PROGRAM DebugMode
VAR
(* Common*)
	d_state: DINT;(*PowerOffState*)
	InitDone:BOOL;
	Busy: BOOL;
	fb_ton: TON;
	PowerState: INT;(*PowerOnState*)
	ton_t: TON;
(*Key Command*)
	LeftTopLinPositionNew:LREAL;
	LeftTopLinVelocityNew:LREAL:=0.02;
	btn_LeftTopLinMove:BOOL;
	btn_LeftTopLinStop:BOOL;
	RightTopLinPositionNew:LREAL;
	RightTopLinVelocityNew:LREAL:=0.02;
	btn_RightTopLinMove:BOOL;
	btn_RightTopLinStop:BOOL;
	LeftBottomLinPositionNew:LREAL;
	LeftBottomLinVelocityNew:LREAL:=0.02;
	btn_LeftBottomLinMove:BOOL;
	btn_LeftBottomLinStop:BOOL;
	RightBottomLinPositionNew:LREAL;
	RightBottomLinVelocityNew:LREAL:=0.02;
	btn_RightBottomLinMove:BOOL;
	btn_RightBottomLinStop:BOOL;
(*LeftTopLin*)
	fb_ton1_1:TON;
	fb_ton1_2:TON;
	LeftTopLinState:DINT;
	LeftTopLinBusy:BOOL;
	LeftTopLin_m_state: DINT;
	LeftTopLin_s_state: DINT;
(*RightTopLin*)
	fb_ton2_1:TON;
	fb_ton2_2:TON;
	RightTopLinState:DINT;
	RightTopLinBusy:BOOL;
	RightTopLin_m_state: DINT;
	RightTopLin_s_state: DINT;
(*LeftBottomLin*)
	fb_ton3_1:TON;
	fb_ton3_2:TON;
	LeftBottomLinState:DINT;
	LeftBottomLinBusy:BOOL;
	LeftBottomLin_m_state: DINT;
	LeftBottomLin_s_state: DINT;
(*RightBottomLin*)
	fb_ton4_1:TON;
	fb_ton4_2:TON;
	RightBottomLinState:DINT;
	RightBottomLinBusy:BOOL;
	RightBottomLin_m_state: DINT;
	RightBottomLin_s_state: DINT;


	btn_LeftTopStop: BOOL;
	(*¼ì²âµ½ÏÞÎ»£¬»Ö¸´Move×´Ì¬*)
	FTrig_ReachLS: F_TRIG;
	FTrig_btn_GapMove: F_TRIG;
	
	RTrig_LeftTopMove:R_TRIG;
	RTrig_RightTopMove:R_TRIG;
	RTrig_LeftBottomMove:R_TRIG;
	RTrig_RightBottomMove:R_TRIG;
	
END_VAR

(*********************************************************************Monitor All Carrirt Position***********************************************)
A_MonitoringAllAxis();
(*********************************************************************A_PosDiffDetection***********************************************)
A_PosDiffDetection();
//
IF st_Power=1 THEN
	InitDone:=TRUE;
END_IF
(*********************************************************************btn_PowerOn************************************************************)
IF btn_Power AND st_Power=0 THEN
	btn_PowerOn:=TRUE;
	btn_Power:=FALSE;
END_IF
IF btn_Power AND st_Power=1 THEN
	btn_PowerOff:=TRUE;
	btn_Power:=FALSE;
END_IF
(*********************************************************************btn_PowerOn************************************************************)
IF btn_PowerOn THEN
	A_PowerOn();
END_IF
(****************************************************ESTOP***********************************************)
IF NOT btn_PowerOff THEN
	IF st_Power=1 AND st_Couple<>0THEN
		Error:=TRUE;
		ErrorID:=101;
		FB_PlcEmergencyStop();
		LED_Error:=TRUE;
	END_IF
END_IF

(*********************************************************************btn_PowerOff************************************************************)
IF btn_PowerOff THEN
	A_PowerOff();
END_IF

A_Motion();
A_CheckTargetPos();


(****************************MoveIndicator***************************)
IF Velo_LeftTopLin>0 THEN
	LeftTopLinMoveIndicator:=1;
ELSIF Velo_LeftTopLin<0 THEN
	LeftTopLinMoveIndicator:=-1;
ELSE
	LeftTopLinMoveIndicator:=0;
END_IF
IF Velo_RightTopLin>0 THEN
	RightTopLinMoveIndicator:=1;
ELSIF Velo_RightTopLin<0 THEN
	RightTopLinMoveIndicator:=-1;
ELSE
	RightTopLinMoveIndicator:=0;
END_IF
IF Velo_LeftBottomLin>0 THEN
	LeftBottomLinMoveIndicator:=1;
ELSIF Velo_LeftBottomLin<0 THEN
	LeftBottomLinMoveIndicator:=-1;
ELSE
	LeftBottomLinMoveIndicator:=0;
END_IF
IF Velo_RightBottomLin>0 THEN
	RightBottomLinMoveIndicator:=1;
ELSIF Velo_RightBottomLin<0 THEN
	RightBottomLinMoveIndicator:=-1;
ELSE
	RightBottomLinMoveIndicator:=0;
END_IF
(*********************************************************************ÏÞÎ»Åö´¥×´Ì¬»Ö¸´************************************************************)
(*Èç¹û¼ì²âµ½ÏØÏÞÎ»¿ª¹ØÏÂ½µÑØ£¬»Ö¸´Move×´Ì¬*)
FTrig_ReachLS(CLK:=Unreach_LS_Far AND Unreach_LS_Near);
IF FTrig_ReachLS.Q THEN
	btn_LeftTopLinStop:=TRUE;
	btn_RightTopLinStop:=TRUE;
	btn_LeftBottomLinStop:=TRUE;
	btn_RightBottomLinStop:=TRUE;
END_IF
IF btn_LeftTopLinStop THEN
	btn_RightTopLinStop:=TRUE;
END_IF
IF btn_RightTopLinStop THEN
	btn_LeftBottomLinStop:=TRUE;
END_IF
IF btn_LeftBottomLinStop THEN
	btn_RightBottomLinStop:=TRUE;
END_IF

IF NOT Unreach_LS_Far AND LeftTopLinPositionNew-Pos_LeftTopLin>0.0005 AND btn_LeftTopLinMove THEN
	btn_LeftTopLinStop:=TRUE;
END_IF
IF NOT Unreach_LS_Near AND RightTopLinPositionNew-Pos_RightTopLin<0.0005 AND btn_RightTopLinMove THEN
	btn_RightTopLinStop:=TRUE;
END_IF
IF NOT Unreach_LS_Far AND LeftBottomLinPositionNew-Pos_LeftBottomLin>0.0005 AND btn_LeftBottomLinMove THEN
	btn_LeftBottomLinStop:=TRUE;
END_IF
IF NOT Unreach_LS_Near AND RightBottomLinPositionNew-Pos_RightBottomLin<0.0005 AND btn_RightBottomLinMove THEN
	btn_RightBottomLinStop:=TRUE;
END_IF

ACTION A_CheckTargetPos:
RTrig_LeftTopMove(CLK:=btn_LeftTopLinMove);
IF RTrig_LeftTopMove.Q THEN
	IF NOT st_Power THEN
			ErrorID:=1501;
			Error:=TRUE;
			ErrorDescription:='Plz PowerOn Frist';
			LED_Error:=TRUE;
			//RETURN;
		ELSIF ABS(LeftTopLinPositionNew-Pos_LeftTopLin)>Threshold_LeftTopPos_Debug THEN
			btn_LeftTopLinStop:=TRUE;
			btn_LeftTopLinMove:=FALSE;
			ErrorID:=1502;
			Error:=TRUE;
			ErrorDescription:='targetPos Out of range!';
			LED_Error:=TRUE;
			//RETURN;
		ELSE
			ErrorID:=0;
			Error:=FALSE;
			ErrorDescription:='';
			LED_Error:=FALSE;
		END_IF
END_IF
RTrig_RightTopMove(CLK:=btn_RightTopLinMove);
IF RTrig_RightTopMove.Q THEN
	IF NOT st_Power THEN
			ErrorID:=1503;
			Error:=TRUE;
			ErrorDescription:='Plz PowerOn Frist';
			LED_Error:=TRUE;
			//RETURN;
		ELSIF ABS(RightTopLinPositionNew-Pos_RightTopLin)>Threshold_RightTopPos_Debug THEN
			btn_RightTopLinStop:=TRUE;
			btn_RightTopLinMove:=FALSE;
			ErrorID:=1504;
			Error:=TRUE;
			ErrorDescription:='targetPos Out of range!';
			LED_Error:=TRUE;
			//RETURN;
		ELSE
			ErrorID:=0;
			Error:=FALSE;
			ErrorDescription:='';
			LED_Error:=FALSE;
		END_IF
END_IF
RTrig_LeftBottomMove(CLK:=btn_LeftBottomLinMove);
IF RTrig_LeftBottomMove.Q THEN
	IF NOT st_Power THEN
			ErrorID:=1505;
			Error:=TRUE;
			ErrorDescription:='Plz PowerOn Frist';
			LED_Error:=TRUE;
			//RETURN;
		ELSIF ABS(LeftBottomLinPositionNew-Pos_LeftBottomLin)>Threshold_LeftBottomPos_Debug THEN
			btn_LeftBottomLinStop:=TRUE;
			btn_LeftBottomLinMove:=FALSE;
			ErrorID:=1506;
			Error:=TRUE;
			ErrorDescription:='targetPos Out of range!';
			LED_Error:=TRUE;
			//RETURN;
		ELSE
			ErrorID:=0;
			Error:=FALSE;
			ErrorDescription:='';
			LED_Error:=FALSE;
		END_IF
END_IF
RTrig_RightBottomMove(CLK:=btn_RightBottomLinMove);
IF RTrig_RightBottomMove.Q THEN
	IF NOT st_Power THEN
			ErrorID:=1507;
			Error:=TRUE;
			ErrorDescription:='Plz PowerOn Frist';
			LED_Error:=TRUE;
			//RETURN;
		ELSIF ABS(RightBottomLinPositionNew-Pos_RightBottomLin)>Threshold_RightBottomPos_Debug THEN
			btn_RightBottomLinStop:=TRUE;
			btn_RightBottomLinMove:=FALSE;
			ErrorID:=1508;
			Error:=TRUE;
			ErrorDescription:='targetPos Out of range!';
			LED_Error:=TRUE;
			//RETURN;
		ELSE
			ErrorID:=0;
			Error:=FALSE;
			ErrorDescription:='';
			LED_Error:=FALSE;
		END_IF
END_IF
END_ACTION

ACTION A_monitoringAllAxis:
(****************************************************************
NAME:			A_MonitoringAllAxis
DATA:			2017.5.8
VERSION:		1.0.0
DESCRIPTION:	

HISTORY:
				2017.5.8	NEW

***************************************************************)

(******************************************************************************************************************************************************)
IF st_power<>0 THEN

IF ABS(Pos_LeftTopLin-Pos_LeftBottomLin)>Threshold_LeftPos_Debug  THEN
		btn_LeftTopLinStop:=TRUE;
		btn_RightTopLinStop:=TRUE;
		btn_LeftBottomLinStop:=TRUE;
		btn_RightBottomLInStop:=TRUE;
		FB_PlcEmergencyStop();
		Error:=TRUE;
		ErrorID:=11;
		LED_Error:=TRUE;
END_IF

IF ABS(Pos_RightTopLin-Pos_RightBottomLin)>Threshold_RightPos_Debug  THEN
		btn_LeftTopLinStop:=TRUE;
		btn_RightTopLinStop:=TRUE;
		btn_LeftBottomLinStop:=TRUE;
		btn_RightBottomLInStop:=TRUE;
		FB_PlcEmergencyStop();
		Error:=TRUE;
		ErrorID:=12;
		LED_Error:=TRUE;
END_IF

IF ABS(Pos_LeftTopLin-Pos_RightTopLin)>Threshold_TopPos_Debug  THEN
		btn_LeftTopLinStop:=TRUE;
		btn_RightTopLinStop:=TRUE;
		btn_LeftBottomLinStop:=TRUE;
		btn_RightBottomLInStop:=TRUE;
		FB_PlcEmergencyStop();
		Error:=TRUE;
		ErrorID:=13;
		LED_Error:=TRUE;
END_IF

IF ABS(Pos_LeftBottomLin-Pos_RightBottomLin)>Threshold_BottomPos_Debug  THEN
		btn_LeftTopLinStop:=TRUE;
		btn_RightTopLinStop:=TRUE;
		btn_LeftBottomLinStop:=TRUE;
		btn_RightBottomLInStop:=TRUE;
		FB_PlcEmergencyStop();
		Error:=TRUE;
		ErrorID:=14;
		LED_Error:=TRUE;
END_IF
END_IF
(*********************************************************************************3.Ã¿Öá¹âÕ¤ºÍ±àÂëÆ÷Î»ÖÃ¶Ô±È¼ì²é**********************************************************************)
END_ACTION

ACTION A_Motion:
(*********************************************************************LeftTop_MOVE*****************************************************************)
//IF InitDone THEN
	IF btn_LeftTopLinMove THEN
		CASE LeftTopLin_m_state OF
			0:
				FB_Move.Mode:=4;					
				FB_Move.CoupleState:=st_Couple;
				FB_Move.PowerState:=st_Power;		
				FB_Move.LeftTopMove:=TRUE;			
				FB_Move.LeftTopPosition:=LeftTopLinPositionNew;
				FB_Move.LeftTopVelocity:=LeftTopLinVelocityNew;	
				FB_Move();								
				LeftTopLin_m_state:=1;
			1:
				FB_Move();
				IF NOT FB_Move.LeftTopDone THEN		
					LeftTopLin_m_state:=1;
					LED_Run:=TRUE;
				ELSE							
					LeftTopLin_m_state:=88;
				END_IF

			88:
				btn_LeftTopLinMove:=FALSE;				
				LeftTopLin_m_state:=0;
				LED_Run:=FALSE;
		END_CASE
	END_IF
//END_IF
(*******************************************************************LeftTop_STOP********************************************************************)
IF btn_LeftTopLinStop OR btn_reset THEN
	LED_Run:=FALSE;
	FB_Move.LeftTopReset:=TRUE;							
	FB_Move();										
	btn_LeftTopLinMove:=FALSE;						
	LeftTopLin_m_state:=0;										
	CASE LeftTopLin_s_state OF
			0:
				FB_Stop.Mode:=4;							
				FB_Stop.CoupleState:=st_Couple;			
				FB_Stop.PowerState:=st_Power;				
				FB_Stop.LeftTopStop:=TRUE;				
				FB_Stop();							
				LeftTopLin_s_state:=1;
			1:
				FB_Stop();
				IF NOT FB_Stop.LeftTopDone THEN		
					LeftTopLin_s_state:=1;
				ELSE								
					LeftTopLin_s_state:=88;
				END_IF
			88:
				btn_LeftTopLinStop:=FALSE;					
				FB_Move.LeftTopReset:=FALSE;				
				LeftTopLin_s_state:=0;
				btn_reset:=FALSE;
		END_CASE

END_IF
(*********************************************************************RightTop_MOVE*****************************************************************)
//IF InitDone THEN
	IF btn_RightTopLinMove THEN
		CASE RightTopLin_m_state OF
			0:
				FB_Move.Mode:=4;						
				FB_Move.CoupleState:=st_Couple;			
				FB_Move.PowerState:=st_Power;			
				FB_Move.RightTopMove:=TRUE;			
				FB_Move.RightTopPosition:=RightTopLinPositionNew;	
				FB_Move.RightTopVelocity:=RightTopLinVelocityNew;	
				FB_Move();								
				RightTopLin_m_state:=1;
			1:
				FB_Move();
				IF NOT FB_Move.RightTopDone THEN		
					RightTopLin_m_state:=1;
					LED_Run:=TRUE;
				ELSE								
					RightTopLin_m_state:=88;
				END_IF

			88:
				btn_RightTopLinMove:=FALSE;				
				RightTopLin_m_state:=0;
				LED_Run:=FALSE;
		END_CASE
	END_IF
//END_IF
(*******************************************************************RightTop_STOP********************************************************************)
IF btn_RightTopLinStop OR btn_reset THEN
	LED_Run:=FALSE;
	FB_Move.RightTopReset:=TRUE;						
	FB_Move();										
	btn_RightTopLinMove:=FALSE;							
	RightTopLin_m_state:=0;										
	CASE RightTopLin_s_state OF
			0:
				FB_Stop.Mode:=4;							
				FB_Stop.CoupleState:=st_Couple;		
				FB_Stop.PowerState:=st_Power;			
				FB_Stop.RightTopStop:=TRUE;				
				FB_Stop();							
				RightTopLin_s_state:=1;
			1:
				FB_Stop();
				IF NOT FB_Stop.RightTopDone THEN			
					RightTopLin_s_state:=1;
				ELSE								
					RightTopLin_s_state:=88;
				END_IF
			88:
				btn_RightTopLinStop:=FALSE;					
				FB_Move.RightTopReset:=FALSE;				
				RightTopLin_s_state:=0;
				btn_reset:=FALSE;
		END_CASE

END_IF
(*********************************************************************LeftBottom_MOVE*****************************************************************)
//IF InitDone THEN
	IF btn_LeftBottomLinMove THEN
		CASE LeftBottomLin_m_state OF
			0:
				FB_Move.Mode:=4;					
				FB_Move.CoupleState:=st_Couple;			
				FB_Move.PowerState:=st_Power;		
				FB_Move.LeftBottomMove:=TRUE;				(*Execute TRUE*)
				FB_Move.LeftBottomPosition:=LeftBottomLinPositionNew;	
				FB_Move.LeftBottomVelocity:=LeftBottomLinVelocityNew;
				FB_Move();								
				LeftBottomLin_m_state:=1;
			1:
				FB_Move();
				IF NOT FB_Move.LeftBottomDone THEN		
					LeftBottomLin_m_state:=1;
					LED_Run:=TRUE;
				ELSE								
					LeftBottomLin_m_state:=88;
				END_IF

			88:
				btn_LeftBottomLinMove:=FALSE;				
				LeftBottomLin_m_state:=0;
				LED_Run:=FALSE;
		END_CASE
	END_IF
//END_IF
(*******************************************************************LeftBottom_STOP********************************************************************)
IF btn_LeftBottomLinStop OR btn_reset THEN
	LED_Run:=FALSE;
	FB_Move.LeftBottomReset:=TRUE;						
	FB_Move();										
	btn_LeftBottomLinMove:=FALSE;						
	LeftBottomLin_m_state:=0;									
	CASE LeftBottomLin_s_state OF
			0:
				FB_Stop.Mode:=4;						
				FB_Stop.CoupleState:=st_Couple;		
				FB_Stop.PowerState:=st_Power;			
				FB_Stop.LeftBottomStop:=TRUE;				
				FB_Stop();						
				LeftBottomLin_s_state:=1;
			1:
				FB_Stop();
				IF NOT FB_Stop.LeftBottomDone THEN			
					LeftBottomLin_s_state:=1;
				ELSE								
					LeftBottomLin_s_state:=88;
				END_IF
			88:
				btn_LeftBottomLinStop:=FALSE;					
				FB_Move.LeftBottomReset:=FALSE;			
				LeftBottomLin_s_state:=0;
				btn_reset:=FALSE;
		END_CASE

END_IF

(*********************************************************************RightTop_MOVE*****************************************************************)
//IF InitDone THEN
	IF btn_RightBottomLinMove THEN
		CASE RightBottomLin_m_state OF
			0:
				FB_Move.Mode:=4;						
				FB_Move.CoupleState:=st_Couple;			
				FB_Move.PowerState:=st_Power;			
				FB_Move.RightBottomMove:=TRUE;				
				FB_Move.RightBottomPosition:=RightBottomLinPositionNew;	
				FB_Move.RightBottomVelocity:=RightBottomLinVelocityNew;	
				FB_Move();								
				RightBottomLin_m_state:=1;
			1:
				FB_Move();
				IF NOT FB_Move.RightBottomDone THEN			
					RightBottomLin_m_state:=1;
					LED_Run:=TRUE;
				ELSE									
					RightBottomLin_m_state:=88;
				END_IF

			88:
				btn_RightBottomLinMove:=FALSE;					
				RightBottomLin_m_state:=0;
				LED_Run:=FALSE;
		END_CASE
	END_IF
//END_IF
(*******************************************************************RightBottom_STOP********************************************************************)
IF btn_RightBottomLinStop OR btn_reset THEN
	LED_Run:=FALSE;
	FB_Move.RightBottomReset:=TRUE;							
	FB_Move();											
	btn_RightBottomLinMove:=FALSE;							
	RightBottomLin_m_state:=0;											
	CASE RightBottomLin_s_state OF
			0:
				FB_Stop.Mode:=4;							
				FB_Stop.CoupleState:=st_Couple;			
				FB_Stop.PowerState:=st_Power;				
				FB_Stop.RightBottomStop:=TRUE;				
				FB_Stop();								
				RightBottomLin_s_state:=1;
			1:
				FB_Stop();
				IF NOT FB_Stop.RightBottomDone THEN			
					RightBottomLin_s_state:=1;
				ELSE									
					RightBottomLin_s_state:=88;
				END_IF
			88:
				btn_RightBottomLinStop:=FALSE;						
				FB_Move.RightBottomReset:=FALSE;				
				RightBottomLin_s_state:=0;
				btn_reset:=FALSE;
		END_CASE

END_IF
END_ACTION

ACTION A_PosDiffDetection:
IF ABS(PosDiff_LeftTopLin_actual-PosDiff_RightTopLin_actual)>0.2 THEN
	ErrorID:=51;
	Error:=TRUE;
	btn_LeftTopLinStop:=TRUE;
	btn_RightTopLinStop:=TRUE;
	btn_LeftBottomLinStop:=TRUE;
	btn_RightBottomLInStop:=TRUE;
	FB_PlcEmergencyStop();
	LED_Error:=TRUE;
ELSIF ABS(PosDiff_LeftBottomLin_actual-PosDiff_RightBottomLin_actual)>0.2 THEN
	ErrorID:=53;
	Error:=TRUE;
	btn_LeftTopLinStop:=TRUE;
	btn_RightTopLinStop:=TRUE;
	btn_LeftBottomLinStop:=TRUE;
	btn_RightBottomLInStop:=TRUE;
	FB_PlcEmergencyStop();
	LED_Error:=TRUE;
END_IF
END_ACTION

ACTION A_PowerOff:
CASE d_state OF
		0:(*PowerOff*)
			FB_Power(Off:=TRUE);
				d_state:=1;
		1:
			IF NOT FB_power.OffStatus THEN
				d_state:=1;
			ELSE
				d_state:=88;
			END_IF
		88:(*ResetAllState*)
			btn_PowerOn:=FALSE;
			btn_PowerOff:=FALSE;
			ton_t.IN:=FALSE;
			InitDone:=FALSE;
			Error:=FALSE;
			ErrorID:=0;
			d_state:=0;

			btn_LeftTopLinMove:=FALSE;
			btn_LeftTopLinStop:=FALSE;
			fb_ton1_1.IN:=FALSE;
			fb_ton1_2.IN:=FALSE;
			LeftTopLinState:=0;
			LeftTopLinBusy:=FALSE;
			LeftTopLin_m_state:=0;
			LeftTopLin_s_state:=0;

			btn_RightTopLinMove:=FALSE;
			btn_RightTopLinStop:=FALSE;
			fb_ton2_1.IN:=FALSE;
			fb_ton2_2.IN:=FALSE;
			RightTopLinState:=0;
			RightTopLinBusy:=FALSE;
			RightTopLin_m_state:=0;
			RightTopLin_s_state:=0;

			btn_LeftBottomLinMove:=FALSE;
			btn_LeftBottomLinStop:=FALSE;
			fb_ton3_1.IN:=FALSE;
			fb_ton3_2.IN:=FALSE;
			LeftBottomLinState:=0;
			LeftBottomLinBusy:=FALSE;
			LeftBottomLin_m_state:=0;
			LeftBottomLin_s_state:=0;

			btn_RightBottomLinMove:=FALSE;
			btn_RightBottomLinStop:=FALSE;
			fb_ton4_1.IN:=FALSE;
			fb_ton4_2.IN:=FALSE;
			RightBottomLinState:=0;
			RightBottomLinBusy:=FALSE;
			RightBottomLin_m_state:=0;
			RightBottomLin_s_state:=0;

		LED_Error:=FALSE;
		LED_Run:=FALSE;

END_CASE
END_ACTION

ACTION A_PowerOn:
(****************************************************************
NAME:			A_SetAxisPositionAndPowerOn
DATA:			2017.3.27
VERSION:		1.0.0
DESCRIPTION:	

HISTORY:
				2017.3.27		NEW
				

***************************************************************)
fb_ton(PT:=t#0.5s);
CASE PowerState OF
	0:	(*FB_Power_On*)
		FB_Power(On:=TRUE);
		fb_ton.IN:=TRUE;
		PowerState:=1;
	1:	(*wait*)
		FB_power();
		IF NOT FB_power.OnStatus THEN		(*FB_Power_OnÃ»ÓÐÖ´ÐÐÍê£¬wait£¬³¬Ê±FB Error*)
			IF NOT fb_ton.Q THEN
				PowerState:=1;
			ELSE
				ErrorID:=1;
				PowerState:=99;
			END_IF
		ELSE
			PowerState:=88;
		END_IF
	88:	(*All Done*)
		btn_PowerOn:=FALSE;
		PowerState:=0;
		Error:=FALSE;
		ErrorID:=0;
		Busy:=FALSE;
		InitDone:=TRUE;
		FB_power.On:=FALSE;
		fb_ton.IN:=FALSE;
	99:
		btn_PowerOn:=FALSE;
		PowerState:=99;
		Error:=TRUE;
		Busy:=FALSE;
		InitDone:=FALSE;
		FB_Power.On:=FALSE;
		fb_ton.IN:=FALSE;
		LED_Error:=TRUE;
END_CASE
END_ACTION

END_PROGRAM

(* stored: Version 1.1.0.1, ProductVersion 3.1.4024.6
   POU DebugMode: Id {9c1b652b-c28b-4723-806b-1a1456d9a5fb}, SpecialFunc None
   Action A_CheckTargetPos: Id {3518206d-5987-427c-af62-ec71343f2283}
   Action A_monitoringAllAxis: Id {d1a34df5-69b1-4771-bf4a-eb30f477489b}
   Action A_Motion: Id {a901098d-045d-4e16-a70b-5dd8d4c69b74}
   Action A_PosDiffDetection: Id {0b914de3-5a16-4135-8c47-916309d8d3da}
   Action A_PowerOff: Id {e677fe86-edfe-48c4-ba29-b932f9bd11d2}
   Action A_PowerOn: Id {3be612a8-046c-45b5-ad28-b2fb90dcb4f1} *)
